{attribute 'linkalways'} 
{attribute 'no_explicit_call' := 'This FB is a CLASS and must be accessed using methods or properties'}
{attribute 'enable_dynamic_creation'}
FUNCTION_BLOCK InputPort EXTENDS Disposable IMPLEMENTS I_InputPort
VAR
	_name : T_MAXSTRING;
	_data : I_Datatype;
	_connectedTo : I_OutputPort;
	parent : I_HostInputPorts;
	eventEmitter : EventEmitter;
	metadataHost : MetadataHost(eventEmitter);
	selfCreatedMetadata : Stack;
END_VAR

METHOD PUBLIC Accept
VAR_INPUT
	Visitor : I_InputPortVisitor;
END_VAR
Visitor.VisitInputPort(THIS^);
metadataHost.Accept(Visitor);
END_METHOD

METHOD PUBLIC AddDataAsMetadata : I_Metadata
VAR_INPUT
	Name : T_MAXSTRING;
	Data : I_Datatype;
END_VAR
VAR
	metadata : I_Metadata;
END_VAR
metadata := CreateMetadata(Name, Data);
selfCreatedMetadata.Push(metadata);
AddDataAsMetadata := metadata;
END_METHOD

METHOD AddMetadata
VAR_INPUT
	Metadata : I_Metadata;
END_VAR
metadataHost.AddMetadata(Metadata);
END_METHOD

PROPERTY PUBLIC Connected : BOOL
GET
Connected := _connectedTo <> 0;
END_GET
END_PROPERTY

METHOD PRIVATE CreateMetadata : I_Metadata
VAR_INPUT
	MetadataName : T_MAXSTRING;
	MetadataData : I_Datatype;
END_VAR
VAR
	pMetadata : POINTER TO Metadata;
END_VAR
pMetadata := __NEW(Metadata(Name := MetadataName, Data := MetadataData, Parent := THIS^));
CreateMetadata := pMetadata^;
END_METHOD

PROPERTY PUBLIC Data : I_Datatype
GET
Data := _data;
END_GET
END_PROPERTY

METHOD PUBLIC Disconnect
IF NOT Connected THEN
	RETURN;
END_IF

_connectedTo.OffEvent('OnOutputPortChanged', THIS^);
_connectedTo := 0;
_data.ClearReference();
END_METHOD

METHOD PROTECTED DisposeSelfCreatedMetadata : BOOL
VAR
	metadata : I_Metadata;
END_VAR
WHILE selfCreatedMetadata.TryPop(metadata) DO
	metadata.Dispose();
END_WHILE
END_METHOD

METHOD PROTECTED EmitOnInputPortChanged
VAR_INPUT
	PortChanged : I_InputPort;
END_VAR
VAR
	pInputPortChangeEvent : POINTER TO InputPortChangedEvent;
END_VAR
pInputPortChangeEvent := __NEW(InputPortChangedEvent(Target := PortChanged));
eventEmitter.Emit('OnInputPortChanged',pInputPortChangeEvent^);
pInputPortChangeEvent^.Dispose();
END_METHOD

METHOD FB_exit : BOOL
VAR_INPUT
	bInCopyCode : BOOL; // if TRUE, the exit method is called for exiting an instance that is copied afterwards (online change).
END_VAR
IF bInCopyCode THEN
	RETURN;
END_IF

DisposeSelfCreatedMetadata();
END_METHOD

METHOD FB_init : BOOL
VAR_INPUT
	bInitRetains : BOOL; // if TRUE, the retain variables are initialized (warm start / cold start)
	bInCopyCode : BOOL;  // if TRUE, the instance afterwards gets moved into the copy code (online change)
	Name : T_MAXSTRING;
	Data : I_Datatype;
	Parent : I_HostInputPorts;
END_VAR
_name := Name;
_data := Data;
RegisterWithParent(Parent);
END_METHOD

METHOD PUBLIC HandleEvent
VAR_INPUT
	Event : I_Event;
END_VAR
VAR
	outputPortChangedEvent : I_OutputPortChangedEvent;
END_VAR
IF __QUERYINTERFACE(Event, outputPortChangedEvent) THEN
	HandleOutputPortChangedEvent(outputPortChangedEvent.Target);
END_IF
END_METHOD

METHOD PROTECTED HandleOutputPortChangedEvent
VAR_INPUT
	Source : I_OutputPort;
END_VAR
EmitOnInputPortChanged(THIS^);
END_METHOD

PROPERTY PUBLIC Name : T_MAXSTRING
GET
Name := _name;
END_GET
END_PROPERTY

METHOD PUBLIC OffEvent
VAR_INPUT
	EventName : T_MaxString;
	EventHandler : I_EventHandler;
END_VAR
eventEmitter.OffEvent(EventName, EventHandler);
END_METHOD

METHOD PUBLIC OnceEvent
VAR_INPUT
	EventName : T_MaxString;
	EventHandler : I_EventHandler;
END_VAR
eventEmitter.OnceEvent(EventName, EventHandler);
END_METHOD

METHOD PUBLIC OnEvent
VAR_INPUT
	EventName : T_MaxString;
	EventHandler : I_EventHandler;
END_VAR
eventEmitter.OnEvent(EventName, EventHandler);
END_METHOD

METHOD PUBLIC RegisterWithParent
VAR_INPUT
	Parent : I_HostInputPorts;
END_VAR
IF Parent = 0 THEN
	RETURN;
END_IF

THIS^.parent := Parent;
Parent.AddInputPort(THIS^);
END_METHOD

METHOD PUBLIC SerializeWith
VAR_INPUT
	Serializer : I_Serializer;
END_VAR
VAR 
	isConnected : BOOL := Connected;
END_VAR
Serializer.StartObject();
Serializer.AddKeyString('name',_name);
Serializer.AddKeyBool('connected',isConnected);
Serializer.Addkey('datatype');
_data.SerializeTypeWith(Serializer);
Serializer.AddkeyObject('value',_data);
metadataHost.SerializeWith(Serializer);
Serializer.EndObject();
END_METHOD

METHOD PUBLIC TryConnectTo : BOOL
VAR_INPUT
	OutputPort : I_OutputPort;
END_VAR
IF NOT _data.TryMakeReferenceOf(OutputPort.Data) THEN
	RETURN;
END_IF

_connectedTo := OutputPort;
_connectedTo.OnEvent('OnOutputPortChanged', THIS^);
TryConnectTo := TRUE;
END_METHOD

METHOD PUBLIC TryGetMetadataByName : BOOL
VAR_INPUT
	Name : T_MAXSTRING;
	Destination : REFERENCE TO I_Metadata;
END_VAR
TryGetMetadataByName := metadataHost.TryGetMetadataByName(Name,Destination);
END_METHOD

END_FUNCTION_BLOCK

(* stored: Version 1.1.0.1, ProductVersion 3.1.4024.12
   POU InputPort: Id {8a76cd64-8399-006f-0213-1bb5b2341bca}, SpecialFunc None
   Folder Constructor: Id {c02273f4-e8fc-0d09-3c19-79f73fa57a1b}
   Folder Destructor: Id {4570fb36-9adb-4191-a9a5-61e46b1d816d}
   Folder Private: Id {1de64b68-f7ef-4fc3-954f-f97872619990}
   Folder Protected: Id {1f1fa75f-3537-0229-2498-8638fd4c140f}
   Method Accept: Id {1625d170-79e2-014d-2c2b-8ace06c47aa1}
   Method AddDataAsMetadata: Id {a5f6d3ba-1b5b-4472-a132-bae6dd8b4cb3}
   Method AddMetadata: Id {285689fb-673d-4cd1-837b-d081f2ca0e5f}
   Property Connected: Id {0eeca197-140f-0917-0914-20aa772b83ae}
   Get Get: Id {7caf9676-d732-0ed2-375f-00350fceb01e}
   Method CreateMetadata: Id {84ecf84e-8734-49bb-9b34-ad514c5ec452}
   Property Data: Id {f697d0c9-35bd-003b-2eed-d1db3a1aaa7d}
   Get Get: Id {9027c130-d714-0b66-2e0c-fed40c3b84cf}
   Method Disconnect: Id {2d2d97fa-faba-033e-23df-3b334614454b}
   Method DisposeSelfCreatedMetadata: Id {1cebc207-eff4-4abd-a1f5-6e19a86ab4c3}
   Method EmitOnInputPortChanged: Id {7ac9cdfd-9dc5-4ff8-8987-c18d9fe1fa6d}
   Method FB_exit: Id {6e882dd7-9d34-4495-b524-7b489ff415e9}
   Method FB_init: Id {85cb6971-3869-03dd-0362-0b78635177f7}
   Method HandleEvent: Id {a301251b-128e-042e-2c82-4ee90daa8459}
   Method HandleOutputPortChangedEvent: Id {9bdbd293-4e3d-0e2f-0079-1e62c2ac0372}
   Property Name: Id {bed621d8-5fb5-029d-2ec1-72a1805573da}
   Get Get: Id {81e0229a-69c1-0712-0a6c-c9c3a3d10c8f}
   Method OffEvent: Id {8831601f-10ed-0308-0255-7aeb488c0bb1}
   Method OnceEvent: Id {02751623-dd18-0013-0361-602d9e5793b3}
   Method OnEvent: Id {6400660c-9990-0d44-03fa-8885dfec75cf}
   Method RegisterWithParent: Id {99f5fd26-21c8-4b31-8e93-5757e5345969}
   Method SerializeWith: Id {baf1e5a1-8726-45d4-a3c3-4b5a88746bac}
   Method TryConnectTo: Id {cf2a22c3-c119-0919-3767-3381d146e55b}
   Method TryGetMetadataByName: Id {9fa16fc6-6579-49be-8cea-0f81ee7da550} *)
